FUNCTION_BLOCK IEEE1451_SENSOR_DISCRETE
  {SET_ATTRIBUTE(OpcUa, SERVICE)}
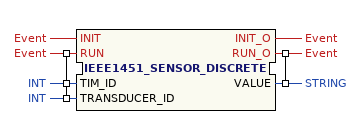
  EVENT_INPUT
    INIT; (* FB Initialization *)
    RUN WITH TRANSDUCER_ID, TIM_ID; (* Read Sensor Request *)
  END_EVENT
  EVENT_OUTPUT
    INIT_O; (* Initialization Confirm *)
    RUN_O WITH VALUE; (* Read Request Confirm *)
  END_EVENT
  VAR_INPUT
    TIM_ID : INT; (* TIM Identification *)
    TRANSDUCER_ID : INT; (* Transducer Identification *)
  END_VAR
  VAR_OUTPUT
    VALUE : STRING; (* Read Result *)
  END_VAR
END_FUNCTION_BLOCK
